FUNCTION_BLOCK Q_SelectColourMap_AUI (* Command Select Colour Map with AUI adapter ( Part 6 - F.60 ) *)
  (* Standard: ISO 11783-6; Description: Copyright (c) 2026 Meisterschulen am Ostbahnhof This program and the accompanying materials are made available under the terms of the Eclipse Public License 2.0 which is available at https://www.eclipse.org/legal/epl-2.0/ SPDX-License-Identifier: EPL-2.0 *)
  (* Version 1.0, 2026-09-11, Franz Höpfinger, Meisterschulen am Ostbahnhof, AUI adapter wrapper for Q_SelectColourMap *)
  PACKAGE isobus::UT::Q;
  (* Documentation:
  Command Select Colour Map with AUI adapter ( Part 6 - F.60 )
   This FB is an AUI adapter wrapper around Q_SelectColourMap.
  *)
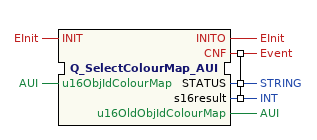
  EVENT_INPUT
    INIT : EInit; (* Service Initialization *)
  END_EVENT
  EVENT_OUTPUT
    INITO : EInit; (* Initialization Confirm *)
    CNF WITH STATUS, s16result; (* Confirmation of Requested Service *)
  END_EVENT
  VAR_OUTPUT
    STATUS : STRING; (* Service Status *)
    s16result : INT; (* retval see description *)
  END_VAR
  SOCKETS
    u16ObjIdColourMap : adapter::types::unidirectional::AUI; (* New object ID of Colour map object *)
  END_SOCKETS
  PLUGS
    u16OldObjIdColourMap : adapter::types::unidirectional::AUI; (* Old object ID of Colour map object *)
  END_PLUGS
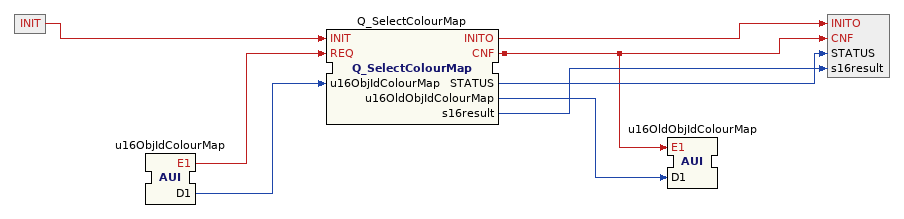
  FBS
    Q_SelectColourMap : isobus::UT::Q::Q_SelectColourMap;
  END_FBS
  EVENT_CONNECTIONS
    INIT TO Q_SelectColourMap.INIT;
    Q_SelectColourMap.INITO TO INITO;
    Q_SelectColourMap.CNF TO CNF;
    u16ObjIdColourMap.E1 TO Q_SelectColourMap.REQ;
    Q_SelectColourMap.CNF TO u16OldObjIdColourMap.E1;
  END_CONNECTIONS
  DATA_CONNECTIONS
    Q_SelectColourMap.STATUS TO STATUS;
    u16ObjIdColourMap.D1 TO Q_SelectColourMap.u16ObjIdColourMap;
    Q_SelectColourMap.u16OldObjIdColourMap TO u16OldObjIdColourMap.D1;
    Q_SelectColourMap.s16result TO s16result;
  END_CONNECTIONS
END_FUNCTION_BLOCK
